TYPE "SpeedMotor_Sts"
VERSION : 0.1
// Block: SpeedMotor_Sts
   STRUCT
      AlarmPresence : Bool;
      WarningPresence : Bool;
      Enabled : Bool;
      Standstill : Bool;
      AtProgrammedSpeed : Bool;
      MoveMinusPermitted : Bool;
      MovePlusPermitted : Bool;
      ActualVelocity : LReal;
   END_STRUCT;

END_TYPE
